{attribute addProperty BoxType "EL7342-0000-0023"}
{attribute addProperty Id "ControlAT %Q*Control_D2752738162"}
{attribute addProperty CRC "1532049156"}
{attribute addProperty SizeInBites "16"}
{attribute addProperty SizeInBytes "2"}
TYPE DCM_Control_Channel_5B513704 :
STRUCT
	{attribute addProperty Name "Control"}
	Control AT %Q* : Control_D2752738;
END_STRUCT
END_TYPE

(* stored: Version 1.2.0.0, ProductVersion 3.1.4024.9
   DUT DCM_Control_Channel_5B513704: Id {2582bdd2-3018-477f-b581-30f7e13dc2ef} *)
